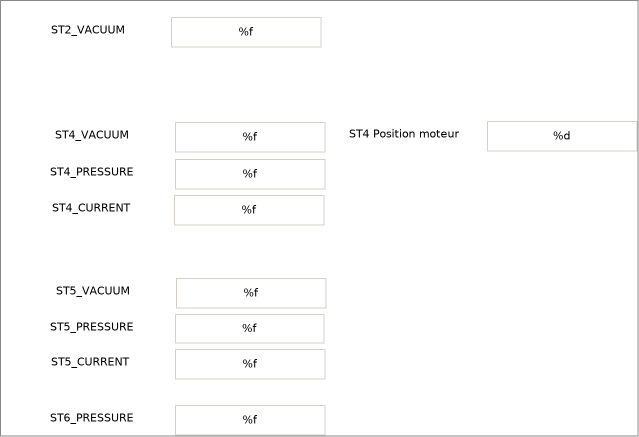
VISUALIZATION AIs  // 639x437
    Textfield (171,17 150x30), "%f", text variable: ST2_VACUUM
    Label (13,15 150x30), "ST2_VACUUM"
    Textfield (175,122 150x30), "%f", text variable: ST4_VACUUM
    Label (17,120 150x30), "ST4_VACUUM"
    Textfield (175,159 150x30), "%f", text variable: ST4_PRESSURE
    Label (17,157 150x30), "ST4_PRESSURE"
    Textfield (176,278 150x30), "%f", text variable: ST5_VACUUM
    Label (18,276 150x30), "ST5_VACUUM"
    Textfield (175,314 149x29), "%f", text variable: ST5_PRESSURE
    Label (17,312 150x30), "ST5_PRESSURE"
    Textfield (175,349 150x30), "%f", text variable: ST5_COURANT
    Label (15,347 150x30), "ST5_CURRENT"
    Textfield (174,195 150x30), "%f", text variable: ST4_COURANT
    Label (16,193 150x30), "ST4_CURRENT"
    Textfield (175,405 150x30), "%f", text variable: ST6_PRESSURE
    Label (17,403 150x30), "ST6_PRESSURE"
    Textfield (487,121 150x30), "%d", text variable: FLAGS.MOTOR_ST4_ACTUAL_POSITION
    Label (329,119 150x30), "ST4 Position moteur"
END_VISUALIZATION

(* stored: Version 1.1.0.1, ProductVersion 3.1.0.26
   Visu AIs: Id {609886ed-1aed-4bde-bdfc-b794a4e5144a} *)
